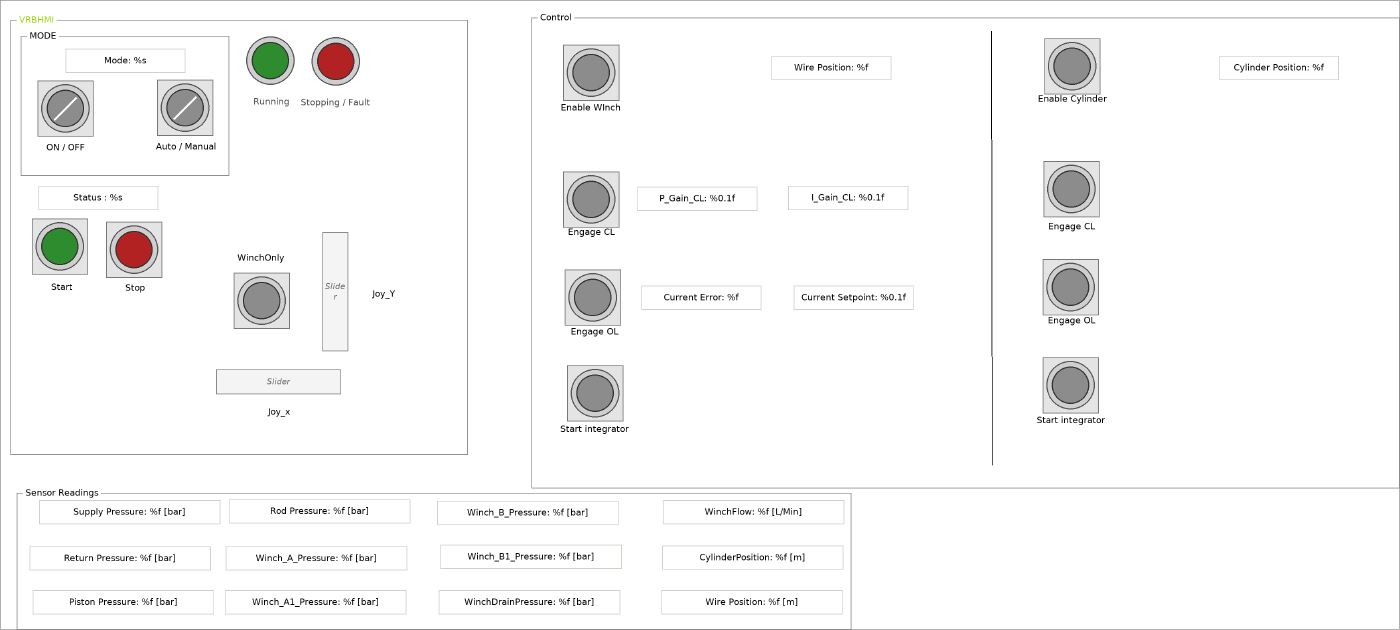
VISUALIZATION VirtualBoxHMI  // 1755x790
    GroupBox (13,17 573x553), "VRBHMI"
        PushSwitch (27,257 70x70), variable: G_Modes.bStart, behaviour: TAP, style: Switch-PushSwitch-Green
        PushSwitch (120,261 70x70), variable: G_Modes.bStop, behaviour: TAP, style: Switch-PushSwitch-Red
        Lamp1 (291,24 70x70), variable: G_Modes.stVisualParams.bRunning, style: Lamp-Lamp1-Green
        Lamp1 (373,25 70x70), variable: G_Modes.stVisualParams.bStop, style: Lamp-Lamp1-Red
        Slider (5682,5127 161x29), scale 0..100
        Slider (5815,4955 30x143), scale 0..100
        Label (5690,5182 150x30), "Joy_X"
        Label (5852,4969 65x118), "Joy_Y"
        Label (360,97 95x29), "Stopping / Fault"
        Label (105,330 103x28), "Stop"
        Label (19,328 91x30), "Start"
        GroupBox (13,20 261x183), "MODE"
            Label (11,133 91x30), "ON / OFF"
            RotarySwitch (171,63 70x70), variable: G_Modes.bAutoMode, behaviour: TOGGLE, style: Switch-RotarySwitch-Gray
            Label (162,132 91x30), "Auto / Manual"
            Textfield (56,24 150x30), "Mode: %s", text variable: G_Modes.eMode
            RotarySwitch (21,64 70x70), variable: G_Modes.bOn, behaviour: TOGGLE, style: Switch-RotarySwitch-Gray
        Textfield (35,216 150x30), "Status : %s", text variable: G_Modes.eStatus
        Label (193,329 103x28)
        Label (280,96 95x29), "Running"
        Slider (258,446 156x31), variable: G_InputsScaled.fJoystickScaledX, scale -1..1
        Slider (391,274 32x149), variable: G_InputsScaled.fJoystickScaledY, scale -1..1
        Label (298,484 78x31), "Joy_x"
        Label (433,338 70x27), "Joy_Y"
        PushSwitch (280,325 70x70), variable: G_Modes.bSwitch, behaviour: TOGGLE, style: Switch-PushSwitch-Gray
        Label (279,293 70x27), "WinchOnly"
    GroupBox (666,14 1089x598), "Control"
        PushSwitch (40,42 70x70), variable: G_Modes.bWinchEnable, behaviour: TOGGLE, style: Switch-PushSwitch-Gray
        Label (29,106 91x30), "Enable WInch"
        PushSwitch (643,34 70x70), variable: G_Modes.bCylEnable, behaviour: TOGGLE, style: Switch-PushSwitch-Gray
        Label (633,95 91x30), "Enable Cylinder"
        PushSwitch (40,201 70x70), variable: G_Modes.stWinchControl.bStartClosedLoop, behaviour: TOGGLE, style: Switch-PushSwitch-Gray
        PushSwitch (42,324 70x70), variable: G_Modes.stWinchControl.bStartFeedForward, behaviour: TOGGLE, style: Switch-PushSwitch-Gray
        PushSwitch (45,444 70x70), variable: G_Modes.stWinchControl.bEnableIntegral, behaviour: TOGGLE, style: Switch-PushSwitch-Gray
        PushSwitch (642,188 70x70), variable: G_Modes.stCylinderControl.bStartClosedLoop, behaviour: TOGGLE, style: Switch-PushSwitch-Gray
        PushSwitch (641,311 70x70), variable: G_Modes.stCylinderControl.bStartFeedForward, behaviour: TOGGLE, style: Switch-PushSwitch-Gray
        PushSwitch (641,434 70x70), variable: G_Modes.stCylinderControl.bEnableIntegral, behaviour: TOGGLE, style: Switch-PushSwitch-Gray
        Label (30,262 91x30), "Engage CL"
        Label (632,255 91x30), "Engage CL"
        Label (34,387 91x30), "Engage OL"
        Label (632,373 91x30), "Engage OL"
        Label (34,509 91x30), "Start integrator"
        Label (631,498 91x30), "Start integrator"
        Line (578,569) (577,25)
        Textfield (301,56 150x30), "Wire Position: %f", text variable: G_InputsScaled.fWirePosition
        Textfield (862,56 150x30), "Cylinder Position: %f", text variable: G_InputsScaled.fCylPosition
        Textfield (133,220 150x30), "P_Gain_CL: %0.1f", text variable: G_Parameters.stControl.stCylControlCloesSettings.fProportionalGain
        Textfield (322,219 150x30), "I_Gain_CL: %0.1f", text variable: G_Parameters.stControl.stCylControlCloesSettings.fIntegralGain
        Textfield (138,344 150x30), "Current Error: %f", text variable: G_ControlParameters.fPosErrorWinch
        Textfield (329,344 150x30), "Current Setpoint: %0.1f", text variable: G_ControlParameters.fVelRefWinch
    GroupBox (21,610 1046x180), "Sensor Readings"
        Textfield (28,17 227x30), "Supply Pressure: %f [bar]", text variable: G_InputsScaled.fSupplyPressure
        Textfield (266,16 227x30), "Rod Pressure: %f [bar]", text variable: G_InputsScaled.fRodPressure
        Textfield (262,75 227x30), "Winch_A_Pressure: %f [bar]", text variable: G_InputsScaled.fWinch_A_Pressure
        Textfield (261,130 227x30), "Winch_A1_Pressure: %f [bar]", text variable: G_InputsScaled.fWinch_A1_Pressure
        Textfield (527,18 227x30), "Winch_B_Pressure: %f [bar]", text variable: G_InputsScaled.fWinch_B_Pressure
        Textfield (531,73 227x30), "Winch_B1_Pressure: %f [bar]", text variable: G_InputsScaled.fWinch_B1_Pressure
        Textfield (529,130 227x30), "WinchDrainPressure: %f [bar]", text variable: G_InputsScaled.fWinchDrainPressure
        Textfield (808,130 227x30), "Wire Position: %f [m]", text variable: G_InputsScaled.fWirePosition
        Textfield (809,74 227x30), "CylinderPosition: %f [m]", text variable: G_InputsScaled.fCylPosition
        Textfield (810,17 227x30), "WinchFlow: %f [L/Min]", text variable: G_InputsScaled.fWinchFlow
        Textfield (16,75 227x30), "Return Pressure: %f [bar]", text variable: G_InputsScaled.fReturnPressure
        Textfield (20,130 227x30), "Piston Pressure: %f [bar]", text variable: G_InputsScaled.fPistonPressure
END_VISUALIZATION

(* stored: Version 1.1.0.1, ProductVersion 3.1.4024.12
   Visu VirtualBoxHMI: Id {86afc6a3-02e3-4d3b-b864-83f52426aa86} *)
